// TIA Portal V20 export
DATA_BLOCK "HmiInterface"   // DB115
// stored: Access Published, MemoryReserve 100, Namespace Unit1.Em12
   VAR
      em : "LAF_typeEmInterface";
      stackNgBox : "LER_typeSequenceInterface";
      cmStackNgBoxDetect : "LBC_typeDigitalSignalInterface";
      cmStackNgBoxFullDetect : "LBC_typeDigitalSignalInterface";
      cmStackNgBoxLoadingUpDown : "LBC_typeTwoWayActuatorInterface";
      cmStackNgBoxUnitMoverBwdFwd : "LBC_typeTwoWayActuatorInterface";
      cmStackNgBoxClampLeftOpenClose : "LBC_typeTwoWayActuatorInterface";
      cmStackNgBoxClampRightOpenClose : "LBC_typeTwoWayActuatorInterface";
      cmStackNgBoxClampMoverOpenClose : "LBC_typeTwoWayActuatorInterface";
      cmStackNgBoxLiftDownUp : "LBC_typeTwoWayActuatorInterface";
      cmStackNgBoxLockDownUp : "LBC_typeTwoWayActuatorInterface";
      intCondition : "Unit1.Em12.typeIntConditionHmiInterface";
   END_VAR
BEGIN
END_DATA_BLOCK
